# EPICS autosave request: iocBoot/generic_motors_ioc/dbSave/XY_P16_.req
%
% BURT Request File
%
% $(P)XY:P16:  X-Y positioner #16
%

file assy.req ASSY=$(P)XY:P16
file mtr1.req MTR1=$(P)XY:mx16
file mtr1.req MTR1=$(P)XY:my16
file drv1.req DRV1=$(P)XY:X16
file drv1.req DRV1=$(P)XY:Y16
